TYPE ST_Position :
STRUCT
	PosX : LREAL;
	PosY: LREAL;
	Initialized: BOOL;
END_STRUCT
END_TYPE

(* stored: Version 1.1.0.1, ProductVersion 3.1.4020.12
   DUT ST_Position: Id {84a5f401-3923-4323-97ca-13218343b32b} *)
